TYPE AX5000_S_0257 :
STRUCT
	Multiplication_factor2:UDINT;
END_STRUCT
END_TYPE

(* stored: Version 1.1.0.1, ProductVersion 3.1.4024.3
   DUT AX5000_S_0257: Id {431392c0-9d24-4edb-b72f-80842ee259d2} *)
